RoboDK station: kr30 cnc 070119 7th axis setup.rdk

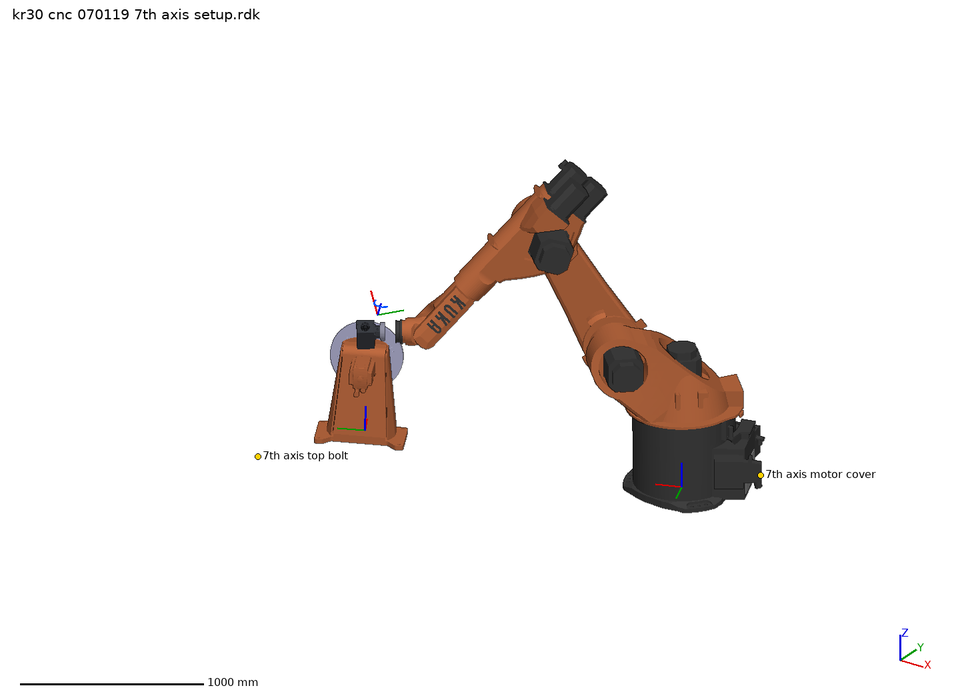
[picture v0: the station drawn from its stored meshes, robots at their saved joint values, targets as dots, program paths as lines]
Station kr30 cnc 070119 7th axis setup. Poses are relative to the parent item; angles as X-Y-Z fixed-axis rotations.
  - frame KUKA KR 30 HA Base at (1535.48, 628.29, -1072.61) mm, rotated rx 0 ry 0 rz -156.31 deg
    - robot KUKA KR 30 HA: 6 axes, payload 30 kg, reach 2033 mm, repeatability 0.05 mm, weight 665 kg
        modified DH rows (alpha deg, a mm, theta deg, d mm): 0, 0, 0, 815; -90, 350, 0, 0; 0, 850, -90, 0; -90, 145, 0, 820; 90, 0, 0, 0; -90, 0, 180, 170
        joint limits [-185, -135, -120, -350, -119, -350] to [185, 35, 158, 350, 119, 350]; home [0, -90, 90, 0, 0, 0]; saved at [-21.518, -62.12, 108.886, 165.582, 46.683, -127.58]
      - tool 1/2" End Mill TCP, TCP at (337.71, -2.2, 160.57) mm, rotated rx 0 ry 90 rz 0 deg, size 415.8 x 102 x 153.6 mm
    - target 7th axis top bolt (joint target) at (1966.13, 1947.63, 927.26) mm, rotated rx -179.2 ry 6.72 rz -171.11 deg; joints [-17.018, -71.525, 110.046, 168.711, 45.865, -170.331, 883.939] of KUKA KR 30 HA
    - target 7th axis motor cover (joint target) at (-417, -111.35, 57.2) mm, rotated rx -135.46 ry -1.69 rz -48.75 deg; joints [-33.388, -54.543, 96.086, 147.711, 45.276, -113.831, 883.939] of KUKA KR 30 HA
  - object box at (500, 500, 500) mm, size 250 x 250 x 250 mm, geometry from box.sld
  - frame KUKA KP1 MD250 Base at (172.34, -439.05, -684.5) mm, rotated rx 2 ry 0.52 rz 120.23 deg
    - robot KUKA KP1 MD250: 1 axes, payload 250 kg
        modified DH rows (alpha deg, a mm, theta deg, d mm): 0, 0, 0, 0
        base shift (70, 10, 428) mm, rotated rx 0 ry 90 rz -2 deg
        joint limits [-180] to [181]; home [0]; saved at [883.939]
      - frame Frame 2 at (0, 0, 500) mm
  - machining project Machining Settings: C:/Users/liqui/Downloads/070119 rotary tower 01.apt | rotZ(0) | rotX(0)*rotY(0) | rotz(0)
  - program Machining (199 instructions, listed below)
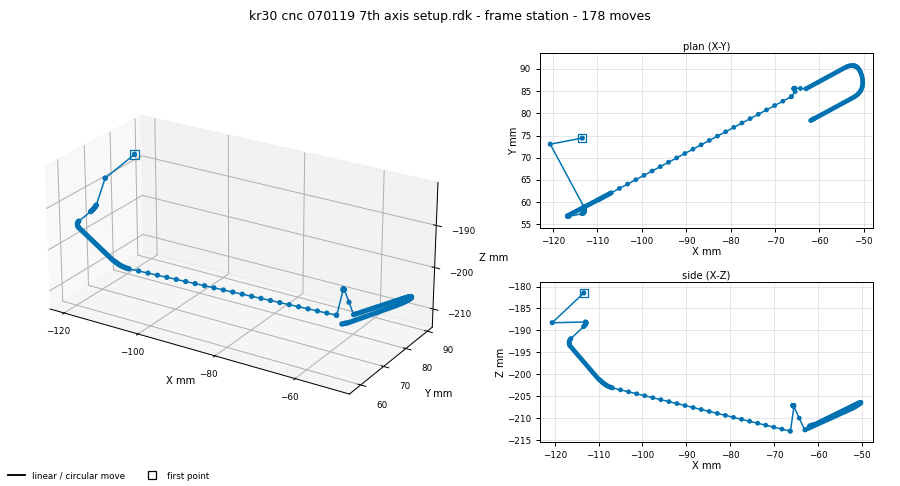
[picture p0: tool path of kr30 cnc 070119 7th axis setup.rdk in frame station, 178 of 178 moves have a stored position in this frame; points joined in program order, loops and branches not executed]

--- program Machining (robot KUKA KR 30 HA) ---
  Smooth(1)
  Set Ref.: Frame 2
  Set Tool: 1/2" End Mill TCP
  Show 1/2" End Mill TCP
  Print: /'1001'
  Print: /''
  Print: /'Flow1'
  Set speed (1000.0 mm/s)
  Set speed (1000.0 mm/s)
  MoveJ 1 to (81.21, 8.78, 12.73) mm, rotated rx 26.94 ry -75.22 rz 32.31 deg; joints [85.605, -66.428, 89.821, -102.377, 79.175, 25.465, 29.968]
  MoveL 2 to (81.21, 8.78, 12.73) mm, rotated rx 26.94 ry -75.22 rz 32.31 deg; joints [85.605, -66.428, 89.821, -102.377, 79.175, 25.465, 29.968]
  MoveL 3 to (76.35, 0.35, 15) mm, rotated rx 26.94 ry -75.22 rz 32.31 deg; joints [85.506, -67.07, 90.729, -102.47, 79.143, 25.749, 29.968]
  MoveL 4 to (76.35, 0.35, 15) mm, rotated rx 26.94 ry -75.22 rz 32.31 deg; joints [85.506, -67.07, 90.729, -102.47, 79.143, 25.749, 29.968]
  Set speed (1000.0 mm/s)
  MoveL 5 to (76.35, 0.35, -0.95) mm, rotated rx 26.94 ry -75.22 rz 32.31 deg; joints [84.968, -66.565, 90.015, -102.666, 78.616, 25.651, 29.968]
  Set speed (16.7 mm/s)
  MoveL 6 to (76.34, 0.33, -1.16) mm, rotated rx 26.93 ry -75.22 rz 32.31 deg; joints [84.961, -66.559, 90.007, -102.668, 78.609, 25.65, 29.968]
  MoveL 7 to (76.31, 0.29, -1.36) mm, rotated rx 26.94 ry -75.22 rz 32.31 deg; joints [84.953, -66.556, 90.003, -102.672, 78.603, 25.651, 29.968]
  MoveL 8 to (76.27, 0.22, -1.55) mm, rotated rx 26.94 ry -75.22 rz 32.31 deg; joints [84.945, -66.554, 90.001, -102.675, 78.595, 25.651, 29.968]
  MoveL 9 to (76.22, 0.12, -1.73) mm, rotated rx 26.94 ry -75.22 rz 32.31 deg; joints [84.937, -66.555, 90.002, -102.679, 78.588, 25.653, 29.968]
  MoveL 10 to (76.15, 0, -1.88) mm, rotated rx 26.93 ry -75.22 rz 32.32 deg; joints [84.929, -66.559, 90.006, -102.681, 78.581, 25.655, 29.968]
  MoveL 11 to (76.07, -0.14, -2.01) mm, rotated rx 26.94 ry -75.22 rz 32.31 deg; joints [84.922, -66.564, 90.014, -102.687, 78.576, 25.66, 29.968]
  MoveL 12 to (75.97, -0.3, -2.11) mm, rotated rx 26.94 ry -75.22 rz 32.3 deg; joints [84.915, -66.571, 90.025, -102.691, 78.571, 25.665, 29.968]
  MoveL 13 to (75.88, -0.47, -2.18) mm, rotated rx 26.94 ry -75.22 rz 32.3 deg; joints [84.909, -66.58, 90.038, -102.695, 78.567, 25.67, 29.968]
  MoveL 14 to (75.78, -0.65, -2.22) mm, rotated rx 26.94 ry -75.22 rz 32.3 deg; joints [84.904, -66.591, 90.053, -102.698, 78.563, 25.676, 29.968]
  MoveL 15 to (75.67, -0.83, -2.22) mm, rotated rx 26.94 ry -75.22 rz 32.3 deg; joints [84.9, -66.603, 90.07, -102.701, 78.561, 25.682, 29.968]
  MoveL 16 to (75.57, -1.01, -2.19) mm, rotated rx 26.94 ry -75.22 rz 32.3 deg; joints [84.898, -66.616, 90.089, -102.703, 78.559, 25.688, 29.968]
  MoveL 17 to (73.64, -4.35, -1.29) mm, rotated rx 26.94 ry -75.22 rz 32.3 deg; joints [84.857, -66.87, 90.448, -102.742, 78.546, 25.801, 29.968]
  MoveL 18 to (73.52, -4.52, -1.24) mm, rotated rx 26.94 ry -75.22 rz 32.3 deg; joints [84.854, -66.884, 90.467, -102.744, 78.545, 25.806, 29.968]
  MoveL 19 to (73.36, -4.68, -1.19) mm, rotated rx 26.94 ry -75.22 rz 32.3 deg; joints [84.852, -66.899, 90.483, -102.745, 78.543, 25.808, 29.968]
  MoveL 20 to (73.19, -4.8, -1.14) mm, rotated rx 26.94 ry -75.22 rz 32.3 deg; joints [84.85, -66.913, 90.497, -102.746, 78.541, 25.808, 29.968]
  MoveL 21 to (72.99, -4.89, -1.1) mm, rotated rx 26.94 ry -75.22 rz 32.3 deg; joints [84.848, -66.927, 90.507, -102.746, 78.539, 25.805, 29.968]
  MoveL 22 to (72.78, -4.94, -1.07) mm, rotated rx 26.94 ry -75.22 rz 32.3 deg; joints [84.847, -66.939, 90.514, -102.746, 78.536, 25.8, 29.968]
  MoveL 23 to (72.56, -4.96, -1.04) mm, rotated rx 26.94 ry -75.22 rz 32.3 deg; joints [84.845, -66.95, 90.516, -102.744, 78.533, 25.791, 29.968]
  MoveL 24 to (72.34, -4.94, -1.02) mm, rotated rx 26.94 ry -75.22 rz 32.3 deg; joints [84.844, -66.959, 90.515, -102.743, 78.53, 25.781, 29.968]
  MoveL 25 to (72.12, -4.88, -1) mm, rotated rx 26.94 ry -75.22 rz 32.3 deg; joints [84.844, -66.966, 90.51, -102.741, 78.527, 25.769, 29.968]
  MoveL 26 to (71.92, -4.78, -1) mm, rotated rx 26.94 ry -75.22 rz 32.3 deg; joints [84.844, -66.971, 90.501, -102.738, 78.523, 25.756, 29.968]
  MoveL 27 to (71.47, -4.52, -1) mm, rotated rx 26.94 ry -75.22 rz 32.3 deg; joints [84.844, -66.98, 90.476, -102.731, 78.516, 25.722, 29.968]
  MoveL 28 to (71.02, -4.26, -1) mm, rotated rx 26.95 ry -75.22 rz 32.3 deg; joints [84.844, -66.988, 90.451, -102.726, 78.509, 25.689, 29.968]
  MoveL 29 to (70.56, -4, -1) mm, rotated rx 26.94 ry -75.22 rz 32.3 deg; joints [84.844, -66.996, 90.425, -102.718, 78.501, 25.655, 29.968]
  MoveL 30 to (70.11, -3.74, -1) mm, rotated rx 26.95 ry -75.22 rz 32.3 deg; joints [84.843, -67.004, 90.4, -102.713, 78.494, 25.622, 29.968]
  MoveL 31 to (69.66, -3.48, -1) mm, rotated rx 26.94 ry -75.22 rz 32.3 deg; joints [84.844, -67.013, 90.374, -102.704, 78.486, 25.588, 29.968]
  MoveL 32 to (69.2, -3.21, -1) mm, rotated rx 26.95 ry -75.22 rz 32.3 deg; joints [84.843, -67.021, 90.349, -102.699, 78.48, 25.555, 29.968]
  MoveL 33 to (68.75, -2.95, -1) mm, rotated rx 26.94 ry -75.22 rz 32.3 deg; joints [84.844, -67.029, 90.324, -102.691, 78.472, 25.521, 29.968]
  MoveL 34 to (68.29, -2.69, -1) mm, rotated rx 26.95 ry -75.22 rz 32.3 deg; joints [84.843, -67.037, 90.298, -102.686, 78.465, 25.488, 29.968]
  MoveL 35 to (67.84, -2.43, -1) mm, rotated rx 26.94 ry -75.22 rz 32.3 deg; joints [84.844, -67.046, 90.273, -102.678, 78.457, 25.454, 29.968]
  MoveL 36 to (67.39, -2.17, -1) mm, rotated rx 26.94 ry -75.22 rz 32.3 deg; joints [84.844, -67.054, 90.247, -102.671, 78.45, 25.421, 29.968]
  MoveL 37 to (66.93, -1.91, -1) mm, rotated rx 26.95 ry -75.22 rz 32.3 deg; joints [84.843, -67.062, 90.222, -102.665, 78.443, 25.388, 29.968]
  MoveL 38 to (66.48, -1.64, -1) mm, rotated rx 27.01 ry -75.91 rz 32.3 deg; joints [84.948, -67.395, 90.525, -102.591, 77.839, 25.403, 29.976]
  MoveL 39 to (66.03, -1.38, -1) mm, rotated rx 27.07 ry -76.61 rz 32.32 deg; joints [85.053, -67.736, 90.836, -102.517, 77.224, 25.416, 29.967]
  MoveL 40 to (65.57, -1.12, -1) mm, rotated rx 27.07 ry -76.61 rz 32.32 deg; joints [85.053, -67.745, 90.81, -102.508, 77.216, 25.382, 29.967]
  MoveL 41 to (65.12, -0.86, -1) mm, rotated rx 27.07 ry -76.61 rz 32.32 deg; joints [85.053, -67.752, 90.784, -102.502, 77.209, 25.349, 29.967]
  MoveL 42 to (64.66, -0.6, -1) mm, rotated rx 27.07 ry -76.61 rz 32.32 deg; joints [85.053, -67.761, 90.758, -102.493, 77.201, 25.314, 29.967]
  MoveL 43 to (64.21, -0.34, -1) mm, rotated rx 27.07 ry -76.61 rz 32.32 deg; joints [85.053, -67.769, 90.732, -102.486, 77.194, 25.28, 29.967]
  MoveL 44 to (63.76, -0.07, -1) mm, rotated rx 27.07 ry -76.61 rz 32.32 deg; joints [85.053, -67.777, 90.707, -102.479, 77.187, 25.247, 29.967]
  MoveL 45 to (63.3, 0.19, -1) mm, rotated rx 27.07 ry -76.61 rz 32.32 deg; joints [85.053, -67.785, 90.681, -102.471, 77.179, 25.212, 29.967]
  MoveL 46 to (62.85, 0.45, -1) mm, rotated rx 27.91 ry -76.51 rz 31.45 deg; joints [85.048, -67.77, 90.716, -102.695, 77.283, 25.31, 29.967]
  MoveL 47 to (62.68, 0.65, -1.02) mm, rotated rx 30.03 ry -76.22 rz 29.27 deg; joints [85.035, -67.709, 90.851, -103.287, 77.568, 25.626, 29.967]
  MoveL 48 to (62.47, 0.8, -1.02) mm, rotated rx 31.69 ry -76.37 rz 25.58 deg; joints [85.115, -67.753, 90.918, -103.645, 77.461, 25.758, 31.991]
  MoveL 49 to (62.27, 0.94, -1.02) mm, rotated rx 33.26 ry -76.55 rz 21.95 deg; joints [85.198, -67.814, 90.984, -103.963, 77.313, 25.866, 34.053]
  MoveL 50 to (62.07, 1.09, -1.02) mm, rotated rx 34.76 ry -76.77 rz 18.36 deg; joints [85.285, -67.895, 91.05, -104.238, 77.122, 25.951, 36.153]
  MoveL 51 to (61.87, 1.25, -1.02) mm, rotated rx 36.18 ry -77.03 rz 14.82 deg; joints [85.375, -67.995, 91.114, -104.467, 76.886, 26.01, 38.29]
  MoveL 52 to (61.67, 1.42, -1.01) mm, rotated rx 37.52 ry -77.33 rz 11.34 deg; joints [85.469, -68.116, 91.178, -104.648, 76.605, 26.042, 40.46]
  MoveL 53 to (61.48, 1.59, -1.01) mm, rotated rx 38.79 ry -77.68 rz 7.9 deg; joints [85.566, -68.257, 91.241, -104.782, 76.276, 26.047, 42.663]
  MoveL 54 to (61.3, 1.77, -1.01) mm, rotated rx 39.98 ry -78.07 rz 4.51 deg; joints [85.665, -68.42, 91.303, -104.861, 75.899, 26.02, 44.893]
  MoveL 55 to (61.12, 1.96, -1.01) mm, rotated rx 41.12 ry -78.51 rz 1.18 deg; joints [85.766, -68.601, 91.366, -104.9, 75.485, 25.969, 47.124]
  MoveL 56 to (60.95, 2.15, -1.01) mm, rotated rx 42.25 ry -78.96 rz -2.12 deg; joints [85.867, -68.796, 91.431, -104.905, 75.044, 25.9, 49.33]
  MoveL 57 to (60.78, 2.35, -1) mm, rotated rx 43.36 ry -79.44 rz -5.35 deg; joints [85.966, -69.004, 91.498, -104.875, 74.578, 25.81, 51.506]
  MoveL 58 to (60.63, 2.55, -1) mm, rotated rx 44.44 ry -79.95 rz -8.53 deg; joints [86.064, -69.225, 91.564, -104.807, 74.087, 25.698, 53.649]
  MoveL 59 to (60.48, 2.76, -1) mm, rotated rx 45.49 ry -80.48 rz -11.64 deg; joints [86.161, -69.458, 91.629, -104.701, 73.573, 25.561, 55.757]
  MoveL 60 to (60.35, 2.97, -1) mm, rotated rx 46.49 ry -81.04 rz -14.67 deg; joints [86.255, -69.7, 91.691, -104.554, 73.037, 25.399, 57.828]
  MoveL 61 to (60.22, 3.19, -1) mm, rotated rx 47.41 ry -81.62 rz -17.58 deg; joints [86.347, -69.952, 91.747, -104.356, 72.477, 25.204, 59.861]
  MoveL 62 to (60.09, 3.41, -1) mm, rotated rx 47.96 ry -83.02 rz -21.97 deg; joints [86.528, -70.493, 91.796, -103.607, 71.206, 24.597, 63.806]
  MoveL 63 to (59.15, 5.32, -1) mm, rotated rx 47.96 ry -83.02 rz -21.97 deg; joints [86.528, -70.522, 91.684, -103.561, 71.173, 24.454, 63.806]
  MoveL 64 to (58.21, 7.24, -1) mm, rotated rx 48 ry -84.15 rz -21.95 deg; joints [86.636, -71.003, 91.844, -102.923, 70.172, 24.001, 63.806]
  MoveL 65 to (57.27, 9.15, -1) mm, rotated rx 48.03 ry -85.17 rz -21.94 deg; joints [86.731, -71.441, 91.973, -102.322, 69.26, 23.551, 63.806]
  MoveL 66 to (56.33, 11.07, -1) mm, rotated rx 48.03 ry -85.17 rz -21.94 deg; joints [86.731, -71.467, 91.858, -102.27, 69.231, 23.404, 63.806]
  MoveL 67 to (55.38, 12.98, -1) mm, rotated rx 48.06 ry -86 rz -21.93 deg; joints [86.805, -71.828, 91.938, -101.756, 68.483, 22.989, 63.806]
  MoveL 68 to (54.44, 14.89, -1) mm, rotated rx 48.08 ry -86.78 rz -21.93 deg; joints [86.872, -72.165, 92, -101.261, 67.785, 22.576, 63.806]
  MoveL 69 to (53.5, 16.81, -1) mm, rotated rx 48.08 ry -86.78 rz -21.93 deg; joints [86.872, -72.189, 91.883, -101.205, 67.758, 22.427, 63.806]
  MoveL 70 to (52.56, 18.72, -1) mm, rotated rx 48.11 ry -87.9 rz -21.94 deg; joints [86.964, -72.657, 92.014, -100.5, 66.776, 21.872, 63.806]
  MoveL 71 to (51.62, 20.64, -1) mm, rotated rx 48.16 ry -88.94 rz -21.98 deg; joints [87.045, -73.093, 92.123, -99.818, 65.862, 21.316, 63.806]
  MoveL 72 to (50.68, 22.55, -1) mm, rotated rx 48.16 ry -88.94 rz -21.97 deg; joints [87.045, -73.116, 92.003, -99.756, 65.838, 21.163, 63.806]
  MoveL 73 to (49.73, 24.47, -1) mm, rotated rx -160.81 ry -90 rz -173 deg; joints [87.124, -73.557, 92.108, -99.038, 64.91, 20.566, 63.815]
  MoveL 74 to (48.79, 26.38, -1) mm, rotated rx -132.01 ry -88.9 rz 158.2 deg; joints [87.2, -74.007, 92.214, -98.278, 63.961, 19.926, 63.806]
  MoveL 75 to (47.85, 28.29, -1) mm, rotated rx -132.01 ry -88.9 rz 158.2 deg; joints [87.2, -74.028, 92.092, -98.21, 63.941, 19.769, 63.806]
  MoveL 76 to (46.91, 30.21, -1) mm, rotated rx -131.98 ry -87.82 rz 158.13 deg; joints [87.271, -74.47, 92.185, -97.429, 63.008, 19.097, 63.825]
  MoveL 77 to (45.97, 32.12, -1) mm, rotated rx -131.98 ry -86.74 rz 158.13 deg; joints [87.337, -74.904, 92.271, -96.634, 62.093, 18.401, 63.806]
  MoveL 78 to (45.03, 34.04, -1) mm, rotated rx -131.98 ry -86.74 rz 158.13 deg; joints [87.337, -74.922, 92.146, -96.559, 62.076, 18.241, 63.806]
  MoveL 79 to (44.08, 35.95, -1) mm, rotated rx -132 ry -85.66 rz 158.09 deg; joints [87.398, -75.356, 92.224, -95.728, 61.161, 17.501, 63.825]
  MoveL 80 to (43.14, 37.87, -1) mm, rotated rx -132.02 ry -84.59 rz 158.09 deg; joints [87.454, -75.78, 92.293, -94.88, 60.266, 16.737, 63.806]
  MoveL 81 to (42.2, 39.78, -1) mm, rotated rx -132.02 ry -84.59 rz 158.09 deg; joints [87.454, -75.797, 92.166, -94.798, 60.254, 16.572, 63.806]
  MoveL 82 to (41.26, 41.69, -1) mm, rotated rx -132.06 ry -83.47 rz 158.04 deg; joints [87.509, -76.24, 92.236, -93.874, 59.321, 15.731, 63.831]
  MoveL 83 to (40.32, 43.61, -1) mm, rotated rx -132.09 ry -82.45 rz 158.04 deg; joints [87.553, -76.634, 92.28, -93.009, 58.491, 14.927, 63.806]
  MoveL 84 to (39.37, 45.52, -1) mm, rotated rx -132.09 ry -82.45 rz 158.04 deg; joints [87.553, -76.648, 92.15, -92.921, 58.484, 14.758, 63.806]
  MoveL 85 to (39.32, 45.63, -1) mm, rotated rx -132.09 ry -82.45 rz 158.04 deg; joints [87.553, -76.649, 92.142, -92.916, 58.483, 14.748, 63.806]
  Set speed (1000.0 mm/s)
  MoveL 86 to (44.74, 48.3, -0.47) mm, rotated rx -132.09 ry -82.45 rz 158.04 deg; joints [87.683, -76.297, 91.706, -92.826, 58.604, 14.642, 63.806]
  Set speed (1000.0 mm/s)
  MoveL 87 to (44.74, 48.3, 0.25) mm, rotated rx -132.09 ry -82.45 rz 158.04 deg; joints [87.71, -76.319, 91.733, -92.821, 58.63, 14.647, 63.806]
  Set speed (1000.0 mm/s)
  MoveL 88 to (44.7, 48.33, 0.25) mm, rotated rx -131.77 ry -80.62 rz 152.83 deg; joints [87.736, -77.135, 91.835, -91.085, 57.155, 12.992, 68.565]
  Set speed (1000.0 mm/s)
  MoveL 89 to (44.66, 48.36, 0.25) mm, rotated rx -130.96 ry -78.72 rz 147.06 deg; joints [87.732, -77.936, 91.867, -89.042, 55.726, 11.066, 73.345]
  Set speed (1000.0 mm/s)
  MoveL 90 to (44.62, 48.4, 0.25) mm, rotated rx -129.91 ry -76.75 rz 141 deg; joints [87.698, -78.71, 91.825, -86.7, 54.377, 8.873, 78.15]
  Set speed (1000.0 mm/s)
  MoveL 91 to (44.58, 48.43, 0.25) mm, rotated rx -128.76 ry -74.74 rz 134.78 deg; joints [87.631, -79.447, 91.711, -84.081, 53.146, 6.429, 82.98]
  Set speed (1000.0 mm/s)
  MoveL 92 to (44.54, 48.46, 0.25) mm, rotated rx -127.59 ry -72.71 rz 128.48 deg; joints [87.534, -80.138, 91.528, -81.215, 52.065, 3.763, 87.839]
  Set speed (1000.0 mm/s)
  MoveL 93 to (44.5, 48.5, 0.25) mm, rotated rx 103.75 ry -34.25 rz -100.57 deg; joints [83.316, -70.414, 103.797, -154.388, 97.57, 51.032, 92.727]
  Set speed (1000.0 mm/s)
  MoveL 94 to (44.46, 48.53, 0.25) mm, rotated rx 104.23 ry -31.2 rz -105.13 deg; joints [82.855, -70.198, 103.971, -156.827, 99.859, 51.88, 97.644]
  Set speed (16.7 mm/s)
  MoveL 95 to (41.57, 48.92, -0.37) mm, rotated rx 104.23 ry -31.2 rz -105.13 deg; joints [82.771, -70.333, 104.157, -156.859, 99.879, 51.965, 97.644]
  MoveL 96 to (38.68, 49.31, -1) mm, rotated rx 104.23 ry -31.2 rz -105.13 deg; joints [82.688, -70.467, 104.342, -156.891, 99.898, 52.05, 97.644]
  MoveL 97 to (38.71, 49.51, -1) mm, rotated rx 104.23 ry -31.2 rz -105.13 deg; joints [82.687, -70.472, 104.334, -156.893, 99.887, 52.044, 97.644]
  MoveL 98 to (38.78, 50.03, -1) mm, rotated rx 104.23 ry -31.2 rz -105.13 deg; joints [82.688, -70.487, 104.314, -156.894, 99.854, 52.031, 97.644]
  MoveL 99 to (38.85, 50.55, -1) mm, rotated rx 104.23 ry -31.2 rz -105.13 deg; joints [82.688, -70.501, 104.295, -156.896, 99.823, 52.017, 97.644]
  MoveL 100 to (38.92, 51.07, -1) mm, rotated rx 104.23 ry -31.2 rz -105.13 deg; joints [82.687, -70.515, 104.274, -156.9, 99.793, 52.004, 97.644]
  MoveL 101 to (38.99, 51.59, -1) mm, rotated rx 104.23 ry -31.2 rz -105.13 deg; joints [82.688, -70.53, 104.255, -156.901, 99.76, 51.99, 97.644]
  MoveL 102 to (39.06, 52.11, -1) mm, rotated rx 104.23 ry -31.2 rz -105.13 deg; joints [82.688, -70.544, 104.235, -156.903, 99.729, 51.976, 97.644]
  MoveL 103 to (39.13, 52.63, -1) mm, rotated rx 104.23 ry -31.2 rz -105.13 deg; joints [82.687, -70.558, 104.215, -156.907, 99.699, 51.963, 97.644]
  MoveL 104 to (39.2, 53.15, -1) mm, rotated rx 104.23 ry -31.2 rz -105.13 deg; joints [82.688, -70.573, 104.195, -156.908, 99.666, 51.949, 97.644]
  MoveL 105 to (39.27, 53.67, -1) mm, rotated rx 104.57 ry -28.24 rz -104.65 deg; joints [82.312, -69.974, 103.994, -159.155, 102.06, 52.567, 97.644]
  MoveL 106 to (39.34, 54.19, -1) mm, rotated rx 104.93 ry -25.29 rz -104.14 deg; joints [81.937, -69.361, 103.706, -161.363, 104.438, 53.091, 97.644]
  MoveL 107 to (39.41, 54.7, -1) mm, rotated rx 104.93 ry -25.3 rz -104.14 deg; joints [81.937, -69.376, 103.688, -161.364, 104.404, 53.08, 97.644]
  MoveL 108 to (39.48, 55.22, -1) mm, rotated rx 104.93 ry -25.3 rz -104.14 deg; joints [81.937, -69.391, 103.668, -161.367, 104.372, 53.069, 97.644]
  MoveL 109 to (39.55, 55.74, -1) mm, rotated rx 104.93 ry -25.3 rz -104.14 deg; joints [81.937, -69.405, 103.649, -161.37, 104.34, 53.058, 97.644]
  MoveL 110 to (39.62, 56.26, -1) mm, rotated rx 104.93 ry -25.29 rz -104.14 deg; joints [81.937, -69.419, 103.629, -161.374, 104.31, 53.047, 97.644]
  MoveL 111 to (39.69, 56.78, -1) mm, rotated rx 104.93 ry -25.3 rz -104.14 deg; joints [81.937, -69.434, 103.611, -161.375, 104.276, 53.035, 97.644]
  MoveL 112 to (39.76, 57.3, -1) mm, rotated rx 104.93 ry -25.3 rz -104.14 deg; joints [81.937, -69.448, 103.591, -161.378, 104.244, 53.024, 97.644]
  MoveL 113 to (39.83, 57.82, -1) mm, rotated rx 104.93 ry -25.29 rz -104.14 deg; joints [81.937, -69.462, 103.571, -161.382, 104.214, 53.013, 97.644]
  MoveL 114 to (39.9, 58.34, -1) mm, rotated rx 104.93 ry -25.3 rz -104.14 deg; joints [81.937, -69.477, 103.552, -161.383, 104.18, 53.002, 97.644]
  MoveL 115 to (39.97, 58.86, -1) mm, rotated rx 104.93 ry -25.3 rz -104.14 deg; joints [81.937, -69.492, 103.533, -161.386, 104.148, 52.991, 97.644]
  MoveL 116 to (40.04, 59.38, -1) mm, rotated rx 104.93 ry -25.29 rz -104.14 deg; joints [81.936, -69.505, 103.513, -161.391, 104.118, 52.98, 97.644]
  MoveL 117 to (40.11, 59.9, -1) mm, rotated rx 105.54 ry -23.97 rz -104.4 deg; joints [81.805, -69.418, 103.583, -162.475, 105.089, 53.51, 97.96]
  MoveL 118 to (40.17, 60.32, -1.01) mm, rotated rx 106.09 ry -27.92 rz -105.65 deg; joints [82.406, -70.659, 104.449, -159.768, 101.591, 53.481, 97.96]
  MoveL 119 to (40.23, 60.71, -1.05) mm, rotated rx 106.89 ry -32.15 rz -107.2 deg; joints [83.043, -72.016, 105.259, -156.888, 97.707, 53.278, 98.016]
  MoveL 120 to (40.3, 61.07, -1.12) mm, rotated rx 108.04 ry -37.04 rz -109.17 deg; joints [83.758, -73.562, 105.972, -153.509, 93.073, 52.721, 98.068]
  MoveL 121 to (40.37, 61.4, -1.21) mm, rotated rx 109.71 ry -42.62 rz -111.75 deg; joints [84.534, -75.275, 106.484, -149.52, 87.641, 51.636, 98.117]
  MoveL 122 to (40.44, 61.7, -1.33) mm, rotated rx 112.23 ry -48.82 rz -115.26 deg; joints [85.336, -77.096, 106.66, -144.776, 81.455, 49.793, 98.163]
  MoveL 123 to (40.52, 61.96, -1.48) mm, rotated rx 115 ry -53.72 rz -118.81 deg; joints [85.915, -78.461, 106.494, -140.67, 76.476, 47.784, 98.207]
  MoveL 124 to (40.56, 62.08, -1.56) mm, rotated rx 117.47 ry -57.1 rz -121.81 deg; joints [86.282, -79.346, 106.206, -137.561, 73.022, 46.046, 98.228]
  MoveL 125 to (40.6, 62.2, -1.65) mm, rotated rx 120.63 ry -60.49 rz -125.51 deg; joints [86.62, -80.182, 105.77, -134.159, 69.557, 43.968, 98.249]
  MoveL 126 to (40.64, 62.3, -1.75) mm, rotated rx 124.7 ry -63.79 rz -130.12 deg; joints [86.919, -80.952, 105.181, -130.443, 66.151, 41.525, 98.27]
  MoveL 127 to (40.68, 62.4, -1.85) mm, rotated rx 129.99 ry -66.93 rz -135.95 deg; joints [87.173, -81.636, 104.445, -126.405, 62.879, 38.703, 98.29]
  MoveL 128 to (40.73, 62.48, -1.96) mm, rotated rx 136.87 ry -69.78 rz -143.36 deg; joints [87.377, -82.223, 103.573, -122.05, 59.818, 35.505, 98.311]
  MoveL 129 to (40.77, 62.56, -2.08) mm, rotated rx 145.71 ry -72.19 rz -152.72 deg; joints [87.528, -82.705, 102.581, -117.401, 57.036, 31.953, 98.332]
  MoveL 130 to (40.81, 62.64, -2.2) mm, rotated rx 156.65 ry -73.99 rz -164.16 deg; joints [87.627, -83.078, 101.494, -112.507, 54.591, 28.095, 98.353]
  MoveL 131 to (40.86, 62.7, -2.33) mm, rotated rx 176.11 ry -75.27 rz 175.64 deg; joints [87.686, -83.44, 99.71, -104.76, 51.622, 21.81, 98.374]
  MoveL 132 to (40.95, 62.8, -2.61) mm, rotated rx -159.63 ry -74.24 rz 150.48 deg; joints [87.616, -83.604, 97.246, -94.435, 49.06, 13.209, 98.418]
  MoveL 133 to (41.05, 62.88, -2.92) mm, rotated rx -142.99 ry -71.34 rz 133.03 deg; joints [87.428, -83.489, 94.802, -84.657, 47.906, 4.939, 98.464]
  MoveL 134 to (41.15, 62.91, -3.25) mm, rotated rx -132.87 ry -67.85 rz 122.18 deg; joints [87.169, -83.191, 92.494, -75.959, 47.823, -2.45, 98.514]
  MoveL 135 to (41.25, 62.92, -3.61) mm, rotated rx -126.62 ry -64.41 rz 115.27 deg; joints [86.879, -82.79, 90.385, -68.559, 48.438, -8.718, 98.566]
  MoveL 136 to (41.36, 62.9, -4) mm, rotated rx -122.58 ry -61.27 rz 110.64 deg; joints [86.584, -82.345, 88.504, -62.429, 49.443, -13.875, 98.623]
  MoveL 137 to (41.47, 62.84, -4.41) mm, rotated rx -119.76 ry -58.39 rz 107.28 deg; joints [86.289, -81.877, 86.792, -57.246, 50.667, -18.194, 98.684]
  MoveL 138 to (41.57, 62.76, -4.82) mm, rotated rx -117.25 ry -55.18 rz 104.18 deg; joints [85.937, -81.283, 84.866, -51.89, 52.352, -22.592, 98.745]
  MoveL 139 to (41.67, 62.65, -5.21) mm, rotated rx -114.96 ry -51.5 rz 101.21 deg; joints [85.506, -80.508, 82.623, -46.258, 54.646, -27.115, 98.803]
  MoveL 140 to (41.75, 62.52, -5.57) mm, rotated rx -112.91 ry -47.34 rz 98.4 deg; joints [84.986, -79.519, 80.035, -40.486, 57.631, -31.609, 98.859]
  MoveL 141 to (41.82, 62.37, -5.9) mm, rotated rx -111.12 ry -42.68 rz 95.77 deg; joints [84.371, -78.284, 77.092, -34.725, 61.35, -35.897, 98.911]
  MoveL 142 to (41.88, 62.19, -6.21) mm, rotated rx -109.61 ry -37.59 rz 93.3 deg; joints [83.662, -76.782, 73.802, -29.123, 65.791, -39.815, 98.962]
  MoveL 143 to (41.93, 61.99, -6.49) mm, rotated rx -108.38 ry -32.13 rz 91.01 deg; joints [82.871, -75.013, 70.207, -23.796, 70.872, -43.228, 99.011]
  MoveL 144 to (41.96, 61.77, -6.74) mm, rotated rx -107.41 ry -26.41 rz 88.88 deg; joints [82.02, -73.001, 66.38, -18.821, 76.448, -46.048, 99.059]
  MoveL 145 to (41.99, 61.53, -6.97) mm, rotated rx -106.7 ry -20.6 rz 86.92 deg; joints [81.142, -70.795, 62.425, -14.233, 82.32, -48.239, 99.107]
  MoveL 146 to (42, 61.26, -7.17) mm, rotated rx -106.22 ry -14.83 rz 85.1 deg; joints [80.27, -68.47, 58.46, -10.031, 88.267, -49.812, 99.154]
  MoveL 147 to (42, 60.97, -7.34) mm, rotated rx -105.93 ry -9.26 rz 83.43 deg; joints [79.437, -66.109, 54.606, -6.189, 94.079, -50.815, 99.202]
  MoveL 148 to (42, 60.65, -7.49) mm, rotated rx -105.82 ry -4.01 rz 81.89 deg; joints [78.669, -63.793, 50.965, -2.672, 99.583, -51.323, 99.251]
  MoveL 149 to (41.97, 60.32, -7.61) mm, rotated rx -105.85 ry 0.84 rz 80.46 deg; joints [77.979, -61.589, 47.611, 0.559, 104.658, -51.417, 99.302]
  MoveL 150 to (41.94, 59.96, -7.7) mm, rotated rx -105.98 ry 5.24 rz 79.15 deg; joints [77.373, -59.546, 44.59, 3.535, 109.237, -51.186, 99.355]
  MoveL 151 to (41.9, 59.58, -7.77) mm, rotated rx -106.19 ry 9.2 rz 77.93 deg; joints [76.85, -57.693, 41.923, 6.281, 113.296, -50.712, 99.41]
  MoveL 152 to (41.84, 59.17, -7.81) mm, rotated rx -106.46 ry 12.71 rz 76.81 deg; joints [76.403, -56.044, 39.608, 8.814, 116.844, -50.067, 99.469]
  MoveL 153 to (41.78, 58.74, -7.82) mm, rotated rx -106.7 ry 13.82 rz 76.31 deg; joints [76.283, -55.603, 39.04, 9.618, 117.91, -49.943, 99.592]
  MoveL 154 to (41.69, 58.23, -7.82) mm, rotated rx -106.13 ry 10.53 rz 77.79 deg; joints [76.66, -57.048, 41.109, 7.238, 114.533, -50.366, 99.182]
  MoveL 155 to (41.61, 57.71, -7.82) mm, rotated rx -106.06 ry 10.88 rz 77.46 deg; joints [76.594, -56.886, 40.908, 7.501, 114.851, -50.234, 99.425]
  MoveL 156 to (41.53, 57.19, -7.82) mm, rotated rx -105.97 ry 11.37 rz 77.52 deg; joints [76.516, -56.615, 40.562, 7.869, 115.308, -50.032, 99.251]
  MoveL 157 to (41.44, 56.68, -7.82) mm, rotated rx -105.89 ry 11.85 rz 77.55 deg; joints [76.44, -56.355, 40.232, 8.23, 115.748, -49.833, 99.109]
  MoveL 158 to (41.36, 56.16, -7.82) mm, rotated rx -105.78 ry 12.44 rz 77.26 deg; joints [76.339, -56.052, 39.831, 8.678, 116.3, -49.589, 99.258]
  MoveL 159 to (41.27, 55.64, -7.82) mm, rotated rx -105.69 ry 12.97 rz 77.13 deg; joints [76.251, -55.776, 39.475, 9.081, 116.783, -49.363, 99.259]
  MoveL 160 to (41.19, 55.13, -7.82) mm, rotated rx -105.6 ry 13.5 rz 77.01 deg; joints [76.163, -55.498, 39.117, 9.493, 117.267, -49.129, 99.26]
  MoveL 161 to (41.11, 54.61, -7.82) mm, rotated rx -105.5 ry 14.07 rz 76.72 deg; joints [76.065, -55.208, 38.738, 9.941, 117.791, -48.876, 99.425]
  MoveL 162 to (41.02, 54.09, -7.82) mm, rotated rx -105.39 ry 14.7 rz 76.74 deg; joints [75.964, -54.859, 38.284, 10.446, 118.374, -48.577, 99.267]
  MoveL 163 to (40.94, 53.57, -7.82) mm, rotated rx -105.33 ry 15.05 rz 76.82 deg; joints [75.91, -54.679, 38.075, 10.723, 118.664, -48.414, 99.11]
  MoveL 164 to (40.85, 53.06, -7.82) mm, rotated rx -104.9 ry 10.94 rz 77.82 deg; joints [76.409, -56.614, 40.834, 7.646, 114.535, -49.262, 99.285]
  MoveL 165 to (40.77, 52.54, -7.82) mm, rotated rx -104.81 ry 11.48 rz 77.7 deg; joints [76.318, -56.332, 40.466, 8.055, 115.033, -49.047, 99.287]
  MoveL 166 to (40.68, 52.02, -7.82) mm, rotated rx -104.73 ry 11.88 rz 77.62 deg; joints [76.25, -56.13, 40.215, 8.361, 115.387, -48.884, 99.284]
  MoveL 167 to (40.6, 51.51, -7.82) mm, rotated rx -104.63 ry 12.47 rz 77.35 deg; joints [76.148, -55.831, 39.82, 8.813, 115.929, -48.643, 99.425]
  MoveL 168 to (40.51, 50.99, -7.82) mm, rotated rx -104.51 ry 13.1 rz 77.34 deg; joints [76.046, -55.495, 39.38, 9.299, 116.502, -48.373, 99.299]
  MoveL 169 to (40.43, 50.47, -7.82) mm, rotated rx -104.45 ry 13.47 rz 77.46 deg; joints [75.988, -55.302, 39.151, 9.589, 116.815, -48.21, 99.11]
  MoveL 170 to (40.35, 49.96, -7.82) mm, rotated rx -104.32 ry 14.18 rz 77.13 deg; joints [75.865, -54.936, 38.661, 10.154, 117.472, -47.894, 99.294]
  MoveL 171 to (40.26, 49.44, -7.82) mm, rotated rx -104.25 ry 14.6 rz 77.05 deg; joints [75.796, -54.73, 38.41, 10.483, 117.823, -47.709, 99.285]
  MoveL 172 to (40.18, 48.92, -7.82) mm, rotated rx -104.16 ry 15.11 rz 77.13 deg; joints [75.714, -54.46, 38.072, 10.894, 118.267, -47.469, 99.11]
  MoveL 173 to (40.09, 48.41, -7.82) mm, rotated rx -104.04 ry 15.49 rz 76.75 deg; joints [75.633, -54.267, 37.824, 11.215, 118.595, -47.244, 99.425]
  MoveL 174 to (40.16, 48.14, -7.8) mm, rotated rx -103.99 ry 14.83 rz 76.92 deg; joints [75.721, -54.585, 38.289, 10.696, 117.934, -47.43, 99.425]
  MoveL 175 to (40.14, 47.89, -7.8) mm, rotated rx -103.7 ry 15.91 rz 78.79 deg; joints [75.565, -53.818, 37.254, 11.609, 118.955, -46.757, 97.393]
  MoveL 176 to (40.12, 47.64, -7.8) mm, rotated rx -103.09 ry 12.27 rz 81.85 deg; joints [76.017, -55.274, 39.358, 8.837, 115.418, -47.319, 95.322]
  MoveL 177 to (40.11, 47.39, -7.8) mm, rotated rx -102.74 ry 13.64 rz 83.73 deg; joints [75.809, -54.36, 38.113, 9.956, 116.729, -46.588, 93.215]
  MoveL 178 to (40.11, 47.14, -7.8) mm, rotated rx -102.39 ry 15.18 rz 85.64 deg; joints [75.575, -53.364, 36.757, 11.24, 118.167, -45.748, 91.072]
